(* IEC 61131-3 sources: com.logicals.lc3.webinar/usRTS_RPMControl_iSOC/src_FB_LIB_SAFE/Bitstring/BYTE, 10 files *)

(* ---- wAND_BYTE_2.iecst ---- *)
NAMESPACE logicals.web.standard
NAMESPACE bitstring

/*
 * Function block wrapper for IEC 61131-3 AND<br>
 * IN1 =  1st value (BYTE)<br>
 * IN2 =  2nd value (BYTE)<br>
 * OUT = IN1 AND IN2 (BYTE)<br>
 */
FUNCTION_BLOCK wAND_BYTE_2
	{ vNameAlignment:="center"; altName:="&"; bgColor:="DodgerBlue"; width:=40; hideIONames; }
	VAR_INPUT
		IN1 : BYTE;
		IN2 : BYTE;
	END_VAR
	VAR_OUTPUT
		OUT: BYTE;
	END_VAR

	OUT := AND(IN1:=IN1, IN2:=IN2, ENO=>ENO);
END_FUNCTION_BLOCK

END_NAMESPACE
END_NAMESPACE

(* ---- wAND_BYTE_3.iecst ---- *)
NAMESPACE logicals.web.standard
NAMESPACE bitstring

/*
 * Function block wrapper for IEC 61131-3 AND<br>
 * IN1 =  1st value (BYTE)<br>
 * IN2 =  2nd value (BYTE)<br>
 * IN3 =  3rd value (BYTE)<br>
 * OUT = IN1 AND IN2 AND IN3 (BYTE)<br>
 */
FUNCTION_BLOCK wAND_BYTE_3
	{ vNameAlignment:="center"; altName:="&"; bgColor:="DodgerBlue"; width:=40; hideIONames; }
	VAR_INPUT
		IN1 : BYTE;
		IN2 : BYTE;
		IN3 : BYTE;
	END_VAR
	VAR_OUTPUT
		OUT: BYTE;
	END_VAR

	OUT := AND(IN1:=IN1, IN2:=IN2, IN3:=IN3, ENO=>ENO);
END_FUNCTION_BLOCK

END_NAMESPACE
END_NAMESPACE

(* ---- wAND_BYTE_4.iecst ---- *)
NAMESPACE logicals.web.standard
NAMESPACE bitstring

/*
 * Function block wrapper for IEC 61131-3 AND<br>
 * IN1 =  1st value (BYTE)<br>
 * IN2 =  2nd value (BYTE)<br>
 * IN3 =  3rd value (BYTE)<br>
 * IN4 =  4th value (BYTE)<br>
 * OUT = IN1 AND IN2 AND IN3 AND IN4 (BYTE)<br>
 */
FUNCTION_BLOCK wAND_BYTE_4
	{ vNameAlignment:="center"; altName:="&"; bgColor:="DodgerBlue"; width:=40; hideIONames; }
	VAR_INPUT
		IN1 : BYTE;
		IN2 : BYTE;
		IN3 : BYTE;
		IN4 : BYTE;
	END_VAR
	VAR_OUTPUT
		OUT: BYTE;
	END_VAR

	OUT := AND(IN1:=IN1, IN2:=IN2, IN3:=IN3, IN4:=IN4, ENO=>ENO);
END_FUNCTION_BLOCK

END_NAMESPACE
END_NAMESPACE

(* ---- wNOT_BYTE.iecst ---- *)
NAMESPACE logicals.web.standard
NAMESPACE bitstring

/*
 * Function block wrapper for IEC 61131-3 NOT<br>
 * IN = input (BYTE)<br>
 * OUT = !IN (BYTE)<br>
 */
FUNCTION_BLOCK wNOT_BYTE
	{ vNameAlignment:="center"; altName:="NOT"; bgColor:="DodgerBlue"; width:=60; hideIONames; }
	VAR_INPUT
		IN : BYTE;
	END_VAR
	VAR_OUTPUT
		OUT: BYTE;
	END_VAR

	OUT := NOT(IN:=IN, ENO=>ENO);
END_FUNCTION_BLOCK

END_NAMESPACE
END_NAMESPACE

(* ---- wOR_BYTE_2.iecst ---- *)
NAMESPACE logicals.web.standard
NAMESPACE bitstring

/*
 * Function block wrapper for IEC 61131-3 OR<br>
 * IN1 =  1st value (BYTE)<br>
 * IN2 =  2nd value (BYTE)<br>
 * OUT = IN1 OR IN2 (BYTE)<br>
 */
FUNCTION_BLOCK wOR_BYTE_2
	{ vNameAlignment:="center"; altName:=">=1"; bgColor:="DodgerBlue"; width:=40; hideIONames; }
	VAR_INPUT
		IN1 : BYTE;
		IN2 : BYTE;
	END_VAR
	VAR_OUTPUT
		OUT: BYTE;
	END_VAR

	OUT := OR(IN1:=IN1, IN2:=IN2, ENO=>ENO);
END_FUNCTION_BLOCK

END_NAMESPACE
END_NAMESPACE

(* ---- wOR_BYTE_3.iecst ---- *)
NAMESPACE logicals.web.standard
NAMESPACE bitstring

/*
 * Function block wrapper for IEC 61131-3 OR<br>
 * IN1 =  1st value (BYTE)<br>
 * IN2 =  2nd value (BYTE)<br>
 * IN3 =  3rd value (BYTE)<br>
 * OUT = IN1 OR IN2 OR IN3 (BYTE)<br>
 */
FUNCTION_BLOCK wOR_BYTE_3
	{ vNameAlignment:="center"; altName:=">=1"; bgColor:="DodgerBlue"; width:=40; hideIONames; }
	VAR_INPUT
		IN1 : BYTE;
		IN2 : BYTE;
		IN3 : BYTE;
	END_VAR
	VAR_OUTPUT
		OUT: BYTE;
	END_VAR

	OUT := OR(IN1:=IN1, IN2:=IN2, IN3:=IN3, ENO=>ENO);
END_FUNCTION_BLOCK

END_NAMESPACE
END_NAMESPACE

(* ---- wOR_BYTE_4.iecst ---- *)
NAMESPACE logicals.web.standard
NAMESPACE bitstring

/*
 * Function block wrapper for IEC 61131-3 OR<br>
 * IN1 =  1st value (BYTE)<br>
 * IN2 =  2nd value (BYTE)<br>
 * IN3 =  3rd value (BYTE)<br>
 * IN4 =  4th value (BYTE)<br>
 * OUT = IN1 OR IN2 OR IN3 OR IN4 (BYTE)<br>
 */
FUNCTION_BLOCK wOR_BYTE_4
	{ vNameAlignment:="center"; altName:=">=1"; bgColor:="DodgerBlue"; width:=40; hideIONames; }
	VAR_INPUT
		IN1 : BYTE;
		IN2 : BYTE;
		IN3 : BYTE;
		IN4 : BYTE;
	END_VAR
	VAR_OUTPUT
		OUT: BYTE;
	END_VAR

	OUT := OR(IN1:=IN1, IN2:=IN2, IN3:=IN3, IN4:=IN4, ENO=>ENO);
END_FUNCTION_BLOCK

END_NAMESPACE
END_NAMESPACE

(* ---- wXOR_BYTE_2.iecst ---- *)
NAMESPACE logicals.web.standard
NAMESPACE bitstring

/*
 * Function block wrapper for IEC 61131-3 XOR<br>
 * IN1 =  1st value (BYTE)<br>
 * IN2 =  2nd value (BYTE)<br>
 * OUT = IN1 XOR IN2 (BYTE)<br>
 */
FUNCTION_BLOCK wXOR_BYTE_2
	{ vNameAlignment:="center"; altName:="=2k+1"; bgColor:="DodgerBlue"; width:=50; hideIONames; }
	VAR_INPUT
		IN1 : BYTE;
		IN2 : BYTE;
	END_VAR
	VAR_OUTPUT
		OUT: BYTE;
	END_VAR

	OUT := XOR(IN1:=IN1, IN2:=IN2, ENO=>ENO);
END_FUNCTION_BLOCK

END_NAMESPACE
END_NAMESPACE

(* ---- wXOR_BYTE_3.iecst ---- *)
NAMESPACE logicals.web.standard
NAMESPACE bitstring

/*
 * Function block wrapper for IEC 61131-3 XOR<br>
 * IN1 =  1st value (BYTE)<br>
 * IN2 =  2nd value (BYTE)<br>
 * IN3 =  3rd value (BYTE)<br>
 * OUT = IN1 XOR IN2 XOR IN3 (BYTE)<br>
 */
FUNCTION_BLOCK wXOR_BYTE_3
	{ vNameAlignment:="center"; altName:="=2k+1"; bgColor:="DodgerBlue"; width:=50; hideIONames; }
	VAR_INPUT
		IN1 : BYTE;
		IN2 : BYTE;
		IN3 : BYTE;
	END_VAR
	VAR_OUTPUT
		OUT: BYTE;
	END_VAR

	OUT := XOR(IN1:=IN1, IN2:=IN2, IN3:=IN3, ENO=>ENO);
END_FUNCTION_BLOCK

END_NAMESPACE
END_NAMESPACE

(* ---- wXOR_BYTE_4.iecst ---- *)
NAMESPACE logicals.web.standard
NAMESPACE bitstring

/*
 * Function block wrapper for IEC 61131-3 XOR<br>
 * IN1 =  1st value (BYTE)<br>
 * IN2 =  2nd value (BYTE)<br>
 * IN3 =  3rd value (BYTE)<br>
 * IN4 =  4th value (BYTE)<br>
 * OUT = IN1 XOR IN2 XOR IN3 XOR IN4 (BYTE)<br>
 */
FUNCTION_BLOCK wXOR_BYTE_4
	{ vNameAlignment:="center"; altName:="=2k+1"; bgColor:="DodgerBlue"; width:=50; hideIONames; }
	VAR_INPUT
		IN1 : BYTE;
		IN2 : BYTE;
		IN3 : BYTE;
		IN4 : BYTE;
	END_VAR
	VAR_OUTPUT
		OUT: BYTE;
	END_VAR

	OUT := XOR(IN1:=IN1, IN2:=IN2, IN3:=IN3, IN4:=IN4, ENO=>ENO);
END_FUNCTION_BLOCK

END_NAMESPACE
END_NAMESPACE
